# EPICS substitutions: transfocatorTest/iocs/BL99I-LCH-IOC-01/BL99I-LCH-IOC-01App/Db/BL99I-LCH-IOC-01_expanded.substitutions
# This file was automatically generated on Wed 07 Nov 2018 14:03:41 GMT from
# source: /home/jjc62351/work/Builder/transfocatorTest/etc/makeIocs/BL99I-LCH-IOC-01.xml
#
# *** Please do not edit this file: edit the source file instead. ***
#

# Macros:
#  P                Device Prefix
#  M                Device Suffix
#  PORT             Delta tau motor controller
#  ADDR             Address on controller
#  DESC             Description, displayed on EDM screen
#  MRES             Motor Step Size (EGU)
#  VELO             Velocity (EGU/s)
#  PREC             Display Precision
#  EGU              Engineering Units
#  TWV              Tweak Step Size (EGU)
#  DTYP             DTYP of record
#  DIR              User Direction
#  VBAS             Base Velocity (EGU/s)
#  VMAX             Max Velocity (EGU/s), defaults to VELO
#  ACCL             Seconds to Velocity
#  BDST             BL Distance (EGU)
#  BVEL             BL Velocity (EGU/s)
#  BACC             BL Seconds to Veloc.
#  DHLM             Dial High Limit
#  DLLM             Dial Low Limit
#  HLM              User High Limit
#  LLM              User Low Limit
#  HLSV             HW Lim. Violation Svr
#  INIT             Startup commands
#  SREV             Steps per Revolution
#  RRES             Readback Step Size (EGU)
#  ERES             Encoder Step Size (EGU)
#  JAR              Jog Acceleration (EGU/s^2)
#  UEIP             Use Encoder If Present
#  URIP             Use RDBL If Present
#  RDBL             Readback Location, set URIP = 1 if you specify this
#  RLNK             Readback output link
#  RTRY             Max retry count
#  DLY              Readback settle time (s)
#  OFF              User Offset (EGU)
#  RDBD             Retry Deadband (EGU)
#  FOFF             Freeze Offset, 0=variable, 1=frozen
#  ADEL             Alarm monitor deadband (EGU)
#  NTM              New Target Monitor, only set to 0 for soft motors
#  FEHIGH           HIGH limit for following error
#  FEHIHI           HIHI limit for following error
#  FEHHSV           HIHI alarm severity for following error
#  FEHSV            HIGH alarm severity for following error
#  SCALE            Scale factor, if pmacSetAxisScale is used this should be set
#  HOMEVIS          If 1 then home is visible on the gui
#  HOMEVISSTR       If HOMEVIS=0, then display this text on the gui instead
#  name             Object name and gui association name
#  alh              Set this to alh to add the motor to the alarm handler and send emails,
#  gda_name         Name to export this as to GDA
#  gda_desc         Description to export this as to GDA
#  SPORT            Delta tau motor controller comms port
#  HOME             Prefix for autohome instance. Defaults to $(P). If unspecified,
#  PMAC             Prefix for pmacStatus instance. Needed to get axis descriptions
#  ALLOW_HOMED_SET  Set to a blank to allow this axis to have its homed
file $(PMACUTIL)/db/dls_pmac_asyn_motor_no_coord.template
{
pattern { P, M, PORT, ADDR, DESC, MRES, VELO, PREC, EGU, TWV, DTYP, DIR, VBAS, VMAX, ACCL, BDST, BVEL, BACC, DHLM, DLLM, HLM, LLM, HLSV, INIT, SREV, RRES, ERES, JAR, UEIP, URIP, RDBL, RLNK, RTRY, DLY, OFF, RDBD, FOFF, ADEL, NTM, FEHIGH, FEHIHI, FEHHSV, FEHSV, SCALE, HOMEVIS, HOMEVISSTR, name, alh, gda_name, gda_desc, SPORT, HOME, PMAC, ALLOW_HOMED_SET }
    { "BL22J-MO-FSWT-01", ":X", "BRICK3", "1", "F-switch X", "0.00005", "1", "5", "mm", "0.1", "asynMotor", "0", "0", "$(VELO)", "0.5", "0", "0", "", "11", "-10", "", "", "MAJOR", "", "1000", "", "", "", "0", "0", "", "", "0", "0", "0", "", "0", "0", "1", "0", "0", "NO_ALARM", "NO_ALARM", "1", "1", "Use motor summary screen", "", "None", "", "$(DESC)", "BRICK3port", "$(P)", "BL22J-MO-STEP-03", "#" }
}
